{attribute 'GeneratedUsingTerminal: EL2262-0000-0001'}
{attribute addProperty BoxType "EL2262-0000-0001"}
{attribute addProperty Id "Output1AT %Q*BOOL1"}
{attribute addProperty CRC "131445834"}
{attribute addProperty Size "1"}
TYPE Sample_07D5B44A EXTENDS OutputBase_10CEE7DE :
STRUCT
	{attribute addProperty Name "Output1"}
	Output1 AT %Q* : BOOL;
END_STRUCT
END_TYPE

(* stored: Version 1.2.0.0, ProductVersion 3.1.4024.11
   DUT Sample_07D5B44A: Id {22c2e7c3-1e0d-4e95-91b3-1cd209cc21b0} *)
